FUNCTION_BLOCK FB_LamparaTemporizada_LD_2
VAR_INPUT
    TiempoEncendido: REAL := 2.0;
    IncrementoTiempo: REAL := 1;    
END_VAR
VAR_OUTPUT
    TiempoPendiente: REAL;
END_VAR
VAR
    Temporizador: TON;

    Memoria: RS;
    Resultado: REAL;
    Tiempo: TIME;
    
    Lampara AT %Q*: BOOL;
    Pulsador AT %I*: BOOL;    
END_VAR

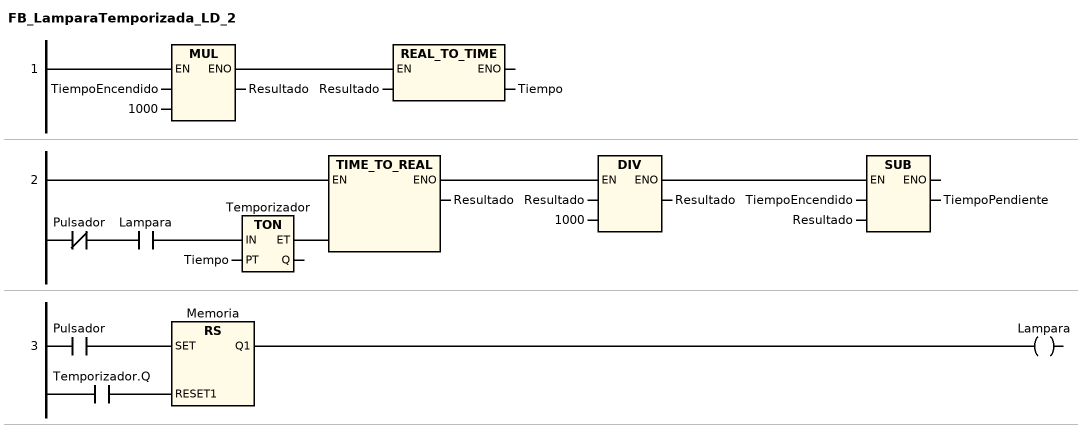
// NETWORK 1
Resultado := TiempoEncendido * 1000;
Tiempo := REAL_TO_TIME(Resultado);

// NETWORK 2
Temporizador(IN := NOT Pulsador AND Lampara, PT := Tiempo); // TON
Resultado := TIME_TO_REAL(Temporizador.ET);
Resultado := Resultado / 1000;
TiempoPendiente := TiempoEncendido - Resultado;

// NETWORK 3
Memoria(SET := Pulsador, RESET1 := Temporizador.Q); // RS
Lampara := Memoria.Q1;

END_FUNCTION_BLOCK

(* stored: Version 1.1.0.1, ProductVersion 3.1.4024.15
   POU FB_LamparaTemporizada_LD_2: Id {5c3eaf1c-4766-4e58-b9c6-070fc8fc3d18}, SpecialFunc None *)
